// TIA Portal V19 export
FUNCTION "APV AHV FP1" : Void   // FC400, STL
{ S7_Optimized_Access := 'TRUE' }
// stored: AutoNumber false
BEGIN

NETWORK
TITLE = **** POLYGON FP1 SWITCHES AND SWINGBEND INTERLOCKS ****
// ? Flowbends are correctly set
      A     "PG_Devices".DI_100_005_X06_X1_3p4;
      AN    "PG_Devices".DI_100_005_X06_X1_3p2;
      =     "Polygon FP1 Route OK";

NETWORK
TITLE = **** HAMBA FP1 SWITCHES AND SWINGBEND INTERLOCKS ****
// Flowbends are correctly set
      AN    "PG_Devices".DI_100_005_X06_X1_3p4;
      A     "PG_Devices".DI_100_005_X06_X1_3p2;
      =     "Hamba FP1 Route OK";

NETWORK
TITLE = **** GASTI FP1 SWITCHES AND SWINGBEND INTERLOCKS ****
// Flowbends are correctly set
      AN    "PG_Devices".DI_100_005_X06_X1_3p4;
      A     "PG_Devices".DI_100_005_X06_X1_3p2;
      =     "Gasti FP1 Route OK";
END_FUNCTION
